{attribute 'qualified_only'}
VAR_GLOBAL CONSTANT
	RecivedBytesBufferSize	:UDINT:=5000;
END_VAR

(* stored: Version 1.1.0.1, ProductVersion 3.1.4026.17
   GVL Param_Supervisor_response: Id {82ace982-3930-44e3-b332-c325fcb8ffd4}, ParameterList True *)
